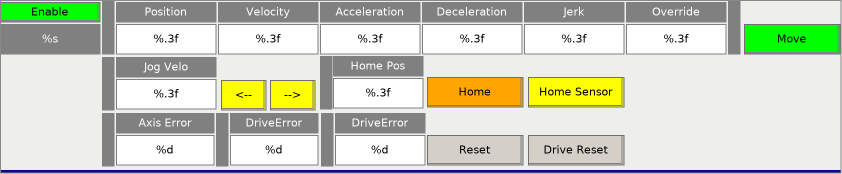
VISUALIZATION VisuAxisControl  // 842x174
VAR_IN_OUT
	sAxisName		: STRING;
	stAxisVisu		: ST_AxisInterface;
END_VAR
    Rectangle (0,24 100x30), "%s", text variable: sAxisName
    Rectangle (116,24 100x30), "%.3f", text variable: stAxisVisu.In.fSetPos
        OnMouseClick: write the text variable via VisuDialogs.Numpad
    Rectangle (116,2 100x20), "Position"
    Rectangle (218,24 100x30), "%.3f", text variable: stAxisVisu.In.fSetVelo
        OnMouseClick: write the text variable via VisuDialogs.Numpad
    Rectangle (218,2 100x20), "Velocity"
    Rectangle (320,24 100x30), "%.3f", text variable: stAxisVisu.In.fSetAcc
        OnMouseClick: write the text variable via VisuDialogs.Numpad
    Rectangle (320,2 100x20), "Acceleration"
    Rectangle (422,24 100x30), "%.3f", text variable: stAxisVisu.In.fSetDec
        OnMouseClick: write the text variable via VisuDialogs.Numpad
    Rectangle (422,2 100x20), "Deceleration"
    Rectangle (524,24 100x30), "%.3f", text variable: stAxisVisu.In.fSetJerk
        OnMouseClick: write the text variable via VisuDialogs.Numpad
    Rectangle (524,2 100x20), "Jerk"
    Rectangle (626,24 100x30), "%.3f", text variable: stAxisVisu.In.fOverride
        OnMouseClick: write the text variable via VisuDialogs.Numpad
    Rectangle (626,2 100x20), "Override"
    Rectangle (116,79 100x30), "%.3f", text variable: stAxisVisu.In.fJogVelo
        OnMouseClick: write the text variable via VisuDialogs.Numpad
    Rectangle (116,57 100x20), "Jog Velo"
    Rectangle (333,78 90x30), "%.3f", text variable: stAxisVisu.In.fHomePos
        OnMouseClick: write the text variable via VisuDialogs.Numpad
    Rectangle (333,56 90x20), "Home Pos"
    Button (0,2 100x20), "Enable"
        toggle stAxisVisu.In.xEnable
    RoundedRectangle (728,1 12x53), colour toggle: stAxisVisu.Out.xMoveDone
    Button (221,80 45x30), "<--"
        tap stAxisVisu.In.xJogBw
    Button (270,80 45x30), "-->"
        tap stAxisVisu.In.xJogFw
    Button (427,77 96x30), "Home"
        toggle stAxisVisu.In.xHome
    Button (528,77 96x30), "Home Sensor"
        toggle stAxisVisu.In.xHomeSensor
    RoundedRectangle (320,56 12x53), colour toggle: stAxisVisu.Out.xHomed
    RoundedRectangle (102,57 12x53)
    RoundedRectangle (102,1 12x53), colour toggle: stAxisVisu.Out.xEnabled
    Button (744,24 96x30), "Move"
        toggle stAxisVisu.In.xMove
    Rectangle (116,135 98x30), "%d", text variable: stAxisVisu.Out.nAxisErrId
    Rectangle (116,113 98x20), "Axis Error"
    RoundedRectangle (102,113 12x53), colour toggle: stAxisVisu.Out.xAxisError
    Rectangle (230,135 88x30), "%d", text variable: stAxisVisu.Out.nDriveErrId
    Rectangle (230,113 88x20), "DriveError"
    RoundedRectangle (216,113 12x53), colour toggle: stAxisVisu.Out.xDriveError
    Rectangle (335,135 90x30), "%d", text variable: stAxisVisu.Out.nFunctionErrId
    Rectangle (335,113 90x20), "DriveError"
    RoundedRectangle (321,113 12x53), colour toggle: stAxisVisu.Out.xFunctionError
    Button (427,135 96x30), "Reset"
        tap stAxisVisu.In.xReset
    Button (528,135 96x30), "Drive Reset"
        tap stAxisVisu.In.xDriveReset
    RoundedRectangle (0,170 840x2)
END_VISUALIZATION

(* stored: Version 1.1.0.1, ProductVersion 3.1.4022.6
   Visu VisuAxisControl: Id {4903126b-5bf0-4578-804c-90bab5cfe7f7} *)
